// TIA Portal V18 program export: 0 tag tables, 2 data types, 1 data blocks, 5 code blocks (in call order from the OBs), 2 instance data blocks

TYPE "User_data_type_1"
// stored: IsFailsafeCompliant false
   STRUCT
      on : Bool;
      off : Bool;
      lamp : Bool;
      pump : Bool;
   END_STRUCT;
END_TYPE

TYPE "User_data_type_2"
// stored: IsFailsafeCompliant false
   STRUCT
      on : Bool;
      off : Bool;
      lamp : Bool;
   END_STRUCT;
END_TYPE

DATA_BLOCK "DB"   // DB1
{ S7_Optimized_Access := 'TRUE' }
VERSION : 0.1
// stored: AutoNumber true, DBAccessibleFromOPCUA true, DBAccessibleFromWebserver true, IsOnlyStoredInLoadMemory false, IsRetainMemResEnabled false, IsWriteProtectedInAS false, MemoryReserve 100
   VAR
      ON : Bool;
      OFF : Bool;
      LAMP : Bool;
      ERROR : Bool;
      STATUS : Word;
      BPOWER : Bool;
   END_VAR
BEGIN
END_DATA_BLOCK

ORGANIZATION_BLOCK "Main"   // OB1, LAD, ProgramCycle
TITLE = "Main Program Sweep (Cycle)"
{ S7_Optimized_Access := 'TRUE' }
VERSION : 0.1
// stored: AutoNumber true, IsIECCheckEnabled false, SetENOAutomatically false
   VAR_INPUT
      Initial_Call : Bool;   // Initial call of this OB
      Remanence : Bool;   // =True, if remanent data are available
   END_VAR
BEGIN

REGION Network 1: sss
END_REGION
END_ORGANIZATION_BLOCK

FUNCTION "Block_1" : Void   // FC1, LAD
{ S7_Optimized_Access := 'TRUE' }
VERSION : 0.1
// stored: AutoNumber true, IsIECCheckEnabled false, SetENOAutomatically false, UDAEnableTagReadback false
BEGIN

REGION Network 1: Network1-addin sss
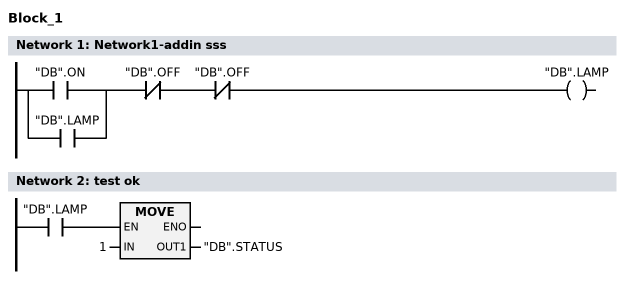
   RUNG wire#powerrail
      Contact( "DB".ON )
      wire#w1
      I_Contact( "DB".OFF )
      I_Contact( "DB".OFF )
      Coil( "DB".LAMP )
   END_RUNG
   RUNG wire#powerrail
      Contact( "DB".LAMP )
   END_RUNG wire#w1
   // the same network as SCL:
   "DB".LAMP := ("DB".ON OR "DB".LAMP) AND NOT "DB".OFF AND NOT "DB".OFF;
END_REGION

REGION Network 2: test ok
   RUNG wire#powerrail
      Contact( "DB".LAMP )
      Move(in := 1, out1 => "DB".STATUS)
   END_RUNG
   // the same network as SCL:
   IF "DB".LAMP THEN "DB".STATUS := 1; END_IF;
END_REGION

REGION Network 3: test
END_REGION
END_FUNCTION

FUNCTION "Block_2" : Void   // FC2, LAD
{ S7_Optimized_Access := 'TRUE' }
VERSION : 0.1
// stored: AutoNumber true, IsIECCheckEnabled false, SetENOAutomatically false, UDAEnableTagReadback false
BEGIN

REGION Network 1: test
END_REGION
END_FUNCTION

FUNCTION_BLOCK "FB1"   // FB1, LAD
{ S7_Optimized_Access := 'TRUE' }
VERSION : 0.1
// stored: AutoNumber true, IsIECCheckEnabled false, IsRetainMemResEnabled false, MemoryReserve 100, SetENOAutomatically false, UDAEnableTagReadback false
BEGIN
END_FUNCTION_BLOCK

FUNCTION_BLOCK "FB2"   // FB2, LAD
{ S7_Optimized_Access := 'TRUE' }
VERSION : 0.1
// stored: AutoNumber true, IsIECCheckEnabled false, IsRetainMemResEnabled false, MemoryReserve 100, SetENOAutomatically false, UDAEnableTagReadback false
BEGIN

REGION Network 1: TEST
END_REGION
END_FUNCTION_BLOCK

DATA_BLOCK "SpeedAxis_1"   // DB2, Motion_DB
// stored: AutoNumber true, DBAccessibleFromOPCUA true, DBAccessibleFromWebserver true, InstanceOfName TO_SpeedAxis, OfSystemLibElement TO_SpeedAxis, OfSystemLibVersion 7.0
TO_SpeedAxis   // technology object, version 7.0
// stored: Connection Interface Actor
// stored: Connection Interface Torque
   // // inherited from TO_Axis
   // // inherited from TO_Object
   // VAR
   //    Velocity { ExternalWritable := 'False'} : LReal;
   //    Acceleration { ExternalWritable := 'False'} : LReal;
   //    ActualSpeed { ExternalWritable := 'False'} : LReal;
   //    VelocitySetpoint { ExternalWritable := 'False'} : LReal;
   //    Actor { S7_SetPoint := 'True'} : TO_Struct_Actor;
   //    TorqueLimiting { S7_SetPoint := 'True'} : TO_Struct_TorqueLimiting;
   //    LoadGear { S7_SetPoint := 'True'} : TO_Struct_LoadGear;
   //    DynamicLimits { S7_SetPoint := 'True'} : TO_Struct_DynamicLimits;
   //    DynamicDefaults { S7_SetPoint := 'True'} : TO_Struct_DynamicDefaults;
   //    Override { S7_SetPoint := 'True'} : TO_Struct_Override;
   //    Units { ExternalWritable := 'False'; S7_SetPoint := 'True'} : TO_Struct_Units;
   //    StatusDrive { ExternalWritable := 'False'; S7_SetPoint := 'True'} : TO_Struct_StatusDrive;
   //    StatusTorqueData { ExternalWritable := 'False'; S7_SetPoint := 'True'} : TO_Struct_StatusTorqueData;
   //    StatusMotionIn { ExternalWritable := 'False'; S7_SetPoint := 'True'} : TO_Struct_StatusMotionIn;
   //    StatusWord { ExternalWritable := 'False'} : DWord;
   //    StatusWord2 { ExternalWritable := 'False'} : DWord;
   //    ErrorWord { ExternalWritable := 'False'} : DWord;
   //    ErrorDetail { ExternalWritable := 'False'; S7_SetPoint := 'True'} : TO_Struct_ErrorDetail;
   //    WarningWord { ExternalWritable := 'False'} : DWord;
   //    ControlPanel { S7_SetPoint := 'True'} : TO_Struct_ControlPanel;
   //    InternalToTrace { S7_SetPoint := 'True'} : Array[1..4] of TO_Struct_Internal;
   //    VirtualAxis { ExternalWritable := 'False'; S7_SetPoint := 'True'} : TO_Struct_VirtualAxis;
   //    Simulation { S7_SetPoint := 'True'} : TO_Struct_AxisSimulation;
   // END_VAR
BEGIN
   DynamicLimits.MaxAcceleration := 1000.0;
   DynamicLimits.MaxDeceleration := 1000.0;
   DynamicLimits.MaxJerk := 20000.0;
   DynamicDefaults.Acceleration := 200.0;
   DynamicDefaults.Deceleration := 200.0;
   DynamicDefaults.Jerk := 4000.0;
   DynamicDefaults.EmergencyDeceleration := 1000.0;
   VirtualAxis.Mode := 1;
   VirtualAxis.Mode := 1;
END_DATA_BLOCK

DATA_BLOCK "SpeedAxis_2"   // DB3, Motion_DB
// stored: AutoNumber true, DBAccessibleFromOPCUA true, DBAccessibleFromWebserver true, InstanceOfName TO_SpeedAxis, OfSystemLibElement TO_SpeedAxis, OfSystemLibVersion 7.0
TO_SpeedAxis   // technology object, version 7.0
// stored: Connection Interface Actor
// stored: Connection Interface Torque
   // // inherited from TO_Axis
   // // inherited from TO_Object
   // VAR
   //    Velocity { ExternalWritable := 'False'} : LReal;
   //    Acceleration { ExternalWritable := 'False'} : LReal;
   //    ActualSpeed { ExternalWritable := 'False'} : LReal;
   //    VelocitySetpoint { ExternalWritable := 'False'} : LReal;
   //    Actor { S7_SetPoint := 'True'} : TO_Struct_Actor;
   //    TorqueLimiting { S7_SetPoint := 'True'} : TO_Struct_TorqueLimiting;
   //    LoadGear { S7_SetPoint := 'True'} : TO_Struct_LoadGear;
   //    DynamicLimits { S7_SetPoint := 'True'} : TO_Struct_DynamicLimits;
   //    DynamicDefaults { S7_SetPoint := 'True'} : TO_Struct_DynamicDefaults;
   //    Override { S7_SetPoint := 'True'} : TO_Struct_Override;
   //    Units { ExternalWritable := 'False'; S7_SetPoint := 'True'} : TO_Struct_Units;
   //    StatusDrive { ExternalWritable := 'False'; S7_SetPoint := 'True'} : TO_Struct_StatusDrive;
   //    StatusTorqueData { ExternalWritable := 'False'; S7_SetPoint := 'True'} : TO_Struct_StatusTorqueData;
   //    StatusMotionIn { ExternalWritable := 'False'; S7_SetPoint := 'True'} : TO_Struct_StatusMotionIn;
   //    StatusWord { ExternalWritable := 'False'} : DWord;
   //    StatusWord2 { ExternalWritable := 'False'} : DWord;
   //    ErrorWord { ExternalWritable := 'False'} : DWord;
   //    ErrorDetail { ExternalWritable := 'False'; S7_SetPoint := 'True'} : TO_Struct_ErrorDetail;
   //    WarningWord { ExternalWritable := 'False'} : DWord;
   //    ControlPanel { S7_SetPoint := 'True'} : TO_Struct_ControlPanel;
   //    InternalToTrace { S7_SetPoint := 'True'} : Array[1..4] of TO_Struct_Internal;
   //    VirtualAxis { ExternalWritable := 'False'; S7_SetPoint := 'True'} : TO_Struct_VirtualAxis;
   //    Simulation { S7_SetPoint := 'True'} : TO_Struct_AxisSimulation;
   // END_VAR
BEGIN
   DynamicLimits.MaxAcceleration := 1000.0;
   DynamicLimits.MaxDeceleration := 1000.0;
   DynamicLimits.MaxJerk := 20000.0;
   DynamicDefaults.Acceleration := 200.0;
   DynamicDefaults.Deceleration := 200.0;
   DynamicDefaults.Jerk := 4000.0;
   DynamicDefaults.EmergencyDeceleration := 1000.0;
   VirtualAxis.Mode := 1;
   VirtualAxis.Mode := 1;
END_DATA_BLOCK
